{attribute 'linkalways'} 
{attribute 'no_explicit_call' := 'This FB is a CLASS and must be accessed using methods or properties'}
{attribute 'enable_dynamic_creation'}
FUNCTION_BLOCK Node_F_VN_GetLayoutInfo EXTENDS VisionNode
VAR
    ipImage : _ITcVnImage;
    aLayoutInfo : _TcVnArray33_UDINT;
    hrPrev : _HRESULT(S_OK);
	hresult : _HRESULT(S_OK);
END_VAR

METHOD PUBLIC  Clone : I_Node
VAR
	pNode : POINTER TO Node_F_VN_GetLayoutInfo;
END_VAR
pNode := __NEW(Node_F_VN_GetLayoutInfo);
Clone := pNode^;
END_METHOD

METHOD FB_init : BOOL
VAR_INPUT
	bInitRetains : BOOL; // if TRUE, the retain variables are initialized (warm start / cold start)
	bInCopyCode : BOOL;  // if TRUE, the instance afterwards gets moved into the copy code (online change)
END_VAR
AddInput('ipImage', ipImage);
AddInput('hrPrev', hrPrev);
AddOutput('aLayoutInfo', aLayoutInfo);
AddOutput('hresult',hresult);
END_METHOD

METHOD PROTECTED OnExecute
hresult.Value := F_VN_GetLayoutInfo(
    ipImage := ipImage.Value,
	aLayoutInfo := aLayoutInfo.Value,
	hrPrev:= hrPrev.Value);
END_METHOD

METHOD PUBLIC PreExecutionCheck
VAR_INPUT
	Check : I_PreExecutionChecks;
END_VAR
Check.IsTrue(ipImage.IsValid, 'ipImage must contain an image');
END_METHOD

END_FUNCTION_BLOCK

(* stored: Version 1.1.0.1, ProductVersion 3.1.4024.13
   POU Node_F_VN_GetLayoutInfo: Id {25cc0df1-996b-0bda-0e6e-57bc753bf9c9}, SpecialFunc None
   Folder Constructor: Id {f1d6b698-8650-00ea-0d2c-dbc5d7872d51}
   Method Clone: Id {ce524958-06f3-0740-3495-c3a824b0bf4f}
   Method FB_init: Id {04a3e386-3333-07fd-3d77-3444de1e989c}
   Method OnExecute: Id {e13566f5-2b45-08b2-1c39-12103f295eaa}
   Method PreExecutionCheck: Id {10ccb412-0f69-0bfe-3240-a57fa87cf269} *)
